// TIA Portal V17 export
// export: Created 2022-12-08T16:45:00.4336249Z, ExportSetting WithDefaults, DisplayName Totally Integrated Automation Portal, DisplayVersion V17 Update 5, DisplayName TIA Portal Openness, DisplayVersion V17 Update 5, DisplayName TIA Portal Version Control Interface, DisplayVersion V17, DisplayName SINAMICS Startdrive Advanced, DisplayVersion V17 SP1, DisplayName SINAMICS Startdrive G130, G150, S120, S150, SINAMICS MV, S210, DisplayVersion V17 SP1, DisplayName SINAMICS Startdrive G110M, G120, G120C, G120D, G120P, G115D, DisplayVersion V17 SP1, DisplayName STEP 7 Professional, DisplayVersion V17 Update 5, DisplayName STEP 7 Safety, DisplayVersion V17, DisplayName WinCC Advanced / Unified PC, DisplayVersion V17 Update 5
FUNCTION "ScalingAnalogInput" : Void   // FC3, LAD
{ S7_Optimized_Access := 'TRUE' }
VERSION : 0.1
// stored: AutoNumber true, IsIECCheckEnabled false, SetENOAutomatically false, UDAEnableTagReadback false
   VAR_INPUT
      RawValue : Int;
   END_VAR
   VAR_OUTPUT
      Output : Real;
   END_VAR
   VAR_TEMP
      Value : Real;
   END_VAR
BEGIN

REGION Network 1
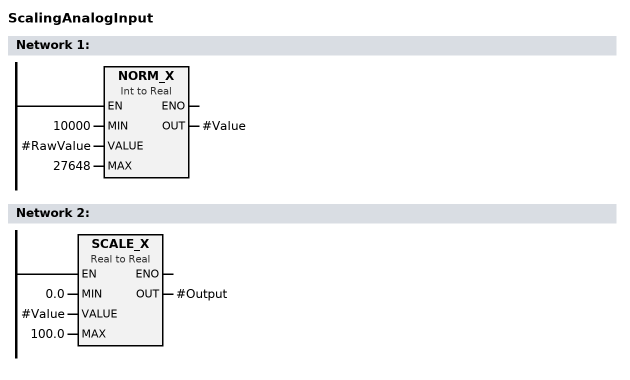
   RUNG wire#powerrail
      { S7_Templates := "[SrcType := Int, DestType := Real]" } Normalize(min := 10000, value := #RawValue, max := 27648, out => #Value)
   END_RUNG
   // the same network as SCL:
   #Value := NORM_X(MIN := 10000, VALUE := #RawValue, MAX := 27648);
END_REGION

REGION Network 2
   RUNG wire#powerrail
      { S7_Templates := "[SrcType := Real, DestType := Real]" } Scale(min := 0.0, value := #Value, max := 100.0, out => #Output)
   END_RUNG
   // the same network as SCL:
   #Output := SCALE_X(MIN := 0.0, VALUE := #Value, MAX := 100.0);
END_REGION
END_FUNCTION
